// TwinCAT 3 PLC project PLC1
// ProgramVersion: 3.1.4024.12
// libraries:
//   Tc2_Standard, * (Beckhoff Automation GmbH)
//   Tc2_System, * (Beckhoff Automation GmbH)
//   Tc3_IPCDiag, * (Beckhoff Automation GmbH)
//   Tc3_JsonXml, * (Beckhoff Automation GmbH)
//   Tc3_Module, * (Beckhoff Automation GmbH)
// project tree:
//   / Class Diagram_Visitor.TcCD (not stored), PlcTask.TcTTO
//   FBs/Exporters/ FB_XmlExporter.TcPOU, FB_SysLogExporter.TcPOU
//   FBs/System Modules/ FB_Conveyor.TcPOU, FB_Heater.TcPOU, FB_IPCDiagnostics.TcPOU
//   ITFs/ I_SysModules.TcIO, I_Visitor.TcIO
//   POUs/ MAIN.TcPOU
// real-time tasks:
//   TASK PlcTask: cycle T#10ms, priority 20, ADS port 350

CONFIGURATION PLC1
    RESOURCE PLC ON TwinCAT3
        TASK PlcTask(INTERVAL := T#10ms, PRIORITY := 20);
        PROGRAM MAIN WITH PlcTask : MAIN;
    END_RESOURCE
END_CONFIGURATION

// ---- ITFs/I_SysModules.TcIO
INTERFACE I_SysModules

METHOD accept
VAR_INPUT
	iVisitor : I_Visitor;
END_VAR
END_METHOD

END_INTERFACE

// ---- ITFs/I_Visitor.TcIO
INTERFACE I_Visitor

METHOD visitConveyor
VAR_INPUT
	fbConveyor : FB_Conveyor;
END_VAR
END_METHOD

METHOD visitHeater
VAR_INPUT
	fbHeater : FB_Heater;
END_VAR
END_METHOD

METHOD visitIPC
VAR_INPUT
	fbIPC : FB_IPCDiagnostics;
END_VAR
END_METHOD

END_INTERFACE

// ---- POUs/MAIN.TcPOU
PROGRAM MAIN
VAR
	// Program Objects
	fbHeater			: ARRAY[0..2] OF FB_Heater;
	fbConveyor 			: ARRAY[0..1] OF FB_Conveyor;
	fbIPCDiagnostics 	: FB_IPCDiagnostics;
	iModules 			: ARRAY[0..5] OF I_SysModules := [fbHeater[0], fbHeater[1], fbHeater[2], fbConveyor[0],  fbConveyor[1], fbIPCDiagnostics];
	
	// Visitor Object Control
	exportVisitor 		: FB_SysLogExporter;
	exportXML			: FB_XmlExporter('C:\TwinCAT\Visitor.xml', 'CX-12345');
	
	// Demo Program Control
	bLogExport			: BOOL;
	bXmlExport			: BOOL;
	bExecSave			: BOOL;
	i					: INT;
END_VAR

// Export the Syslog
IF bLogExport THEN
	bLogExport := FALSE;
	FOR i := 0 TO 5 DO
		iModules[i].accept(exportVisitor);
	END_FOR
END_IF

// Export for XML
IF bXmlExport THEN
	bXmlExport := FALSE;
	FOR i := 0 TO 5 DO
		iModules[i].accept(exportXML);
	END_FOR
	bExecSave := TRUE;
END_IF

IF exportXML.saveDoc(bExec := bExecSave) THEN
	bExecSave := FALSE;
END_IF

END_PROGRAM

// ---- FBs/System Modules/FB_Heater.TcPOU
{attribute 'reflection'} 
FUNCTION_BLOCK FB_Heater IMPLEMENTS I_SysModules
VAR
	lrCurrentTemp : LREAL := 72.0;
	sStatus		  : STRING := 'Heating...';
	
	{attribute 'instance-path'} 
    {attribute 'noinit'} 
    sPath : STRING; 
END_VAR

METHOD accept
VAR_INPUT
	iVisitor : I_Visitor;
END_VAR
iVisitor.visitHeater(THIS^);
END_METHOD

PROPERTY pPath : STRING
GET
pPath := THIS^.sPath;
END_GET
END_PROPERTY

PROPERTY pStatus : STRING
GET
pStatus := THIS^.sStatus;
END_GET
END_PROPERTY

PROPERTY pTemp : LREAL
GET
pTemp := THIS^.lrCurrentTemp;
END_GET
END_PROPERTY

END_FUNCTION_BLOCK

// ---- FBs/System Modules/FB_Conveyor.TcPOU
{attribute 'reflection'} 
FUNCTION_BLOCK FB_Conveyor IMPLEMENTS I_SysModules
VAR
	lrVelocity 	: LREAL := 500.00;
	lrPosition 	: LREAL := 127.00;
	sStatus		: STRING := 'Running';
	
	{attribute 'instance-path'} 
    {attribute 'noinit'} 
    sPath : STRING; 
END_VAR

METHOD accept
VAR_INPUT
	iVisitor : I_Visitor;
END_VAR
iVisitor.visitConveyor(THIS^);
END_METHOD

PROPERTY pPath : STRING
GET
pPath := THIS^.sPath;
END_GET
END_PROPERTY

PROPERTY pPosition : LREAL
GET
pPosition := THIS^.lrPosition;
END_GET
END_PROPERTY

PROPERTY pStatus : STRING
GET
pStatus := THIS^.sStatus;
END_GET
END_PROPERTY

PROPERTY pVelocity : LREAL
GET
pVelocity := THIS^.lrPosition;
END_GET
END_PROPERTY

END_FUNCTION_BLOCK

// ---- FBs/System Modules/FB_IPCDiagnostics.TcPOU
{attribute 'reflection'} 
FUNCTION_BLOCK FB_IPCDiagnostics IMPLEMENTS I_SysModules
VAR
	nCpuTemperature	: INT := 75;	// CPU temperature [°F]
	nCpuUsage       : INT := 5;    // CPU usage [%]
	
	
	{attribute 'instance-path'} 
    {attribute 'noinit'} 
    sPath : STRING; 
END_VAR

METHOD accept
VAR_INPUT
	iVisitor : I_Visitor;
END_VAR
iVisitor.visitIPC(THIS^);
END_METHOD

PROPERTY pCPU_Temp : INT
GET
pCPU_Temp := THIS^.nCpuTemperature;
END_GET
END_PROPERTY

PROPERTY pCPU_Usage : INT
GET
pCPU_Usage := THIS^.nCpuUsage;
END_GET
END_PROPERTY

PROPERTY pPath : STRING
GET
pPath := THIS^.sPath;
END_GET
END_PROPERTY

END_FUNCTION_BLOCK

// ---- FBs/Exporters/FB_SysLogExporter.TcPOU
FUNCTION_BLOCK FB_SysLogExporter IMPLEMENTS I_Visitor
VAR_INPUT
END_VAR
VAR_OUTPUT
END_VAR
VAR
END_VAR

METHOD visitConveyor
VAR_INPUT
	fbConveyor : FB_Conveyor;
END_VAR
ADSLOGSTR( msgCtrlMask := ADSLOG_MSGTYPE_LOG, msgFmtStr := '', strArg := '');
ADSLOGSTR( msgCtrlMask := ADSLOG_MSGTYPE_LOG, msgFmtStr := 'PLC Msg. *** Printing Messages For: %s', strArg := fbConveyor.pPath);
ADSLOGSTR( msgCtrlMask := ADSLOG_MSGTYPE_LOG, msgFmtStr := CONCAT(fbConveyor.pPath,':: Status := %s'), strArg := TO_STRING(fbConveyor.pStatus));
ADSLOGSTR( msgCtrlMask := ADSLOG_MSGTYPE_LOG, msgFmtStr := CONCAT(fbConveyor.pPath,':: Velocity := %s'), strArg := TO_STRING(fbConveyor.pVelocity));
ADSLOGSTR( msgCtrlMask := ADSLOG_MSGTYPE_LOG, msgFmtStr := CONCAT(fbConveyor.pPath,':: Position := %s'), strArg := TO_STRING(fbConveyor.pPosition));
END_METHOD

METHOD visitHeater
VAR_INPUT
	fbHeater : FB_Heater;
END_VAR
ADSLOGSTR( msgCtrlMask := ADSLOG_MSGTYPE_LOG, msgFmtStr := '', strArg := '');
ADSLOGSTR( msgCtrlMask := ADSLOG_MSGTYPE_LOG, msgFmtStr := 'PLC Msg. *** Printing Messages For: %s', strArg := fbHeater.pPath);
ADSLOGSTR( msgCtrlMask := ADSLOG_MSGTYPE_LOG, msgFmtStr := CONCAT(fbHeater.pPath,':: Status := %s'), strArg := TO_STRING(fbHeater.pStatus));
ADSLOGSTR( msgCtrlMask := ADSLOG_MSGTYPE_LOG, msgFmtStr := CONCAT(fbHeater.pPath,':: Temperature := %s'), strArg := TO_STRING(fbHeater.pTemp));
END_METHOD

METHOD visitIPC
VAR_INPUT
	fbIPC : FB_IPCDiagnostics;
END_VAR
ADSLOGSTR( msgCtrlMask := ADSLOG_MSGTYPE_LOG, msgFmtStr := '', strArg := '');
ADSLOGSTR( msgCtrlMask := ADSLOG_MSGTYPE_LOG, msgFmtStr := 'PLC Msg. *** Printing Messages For: %s', strArg := fbIPC.pPath);
ADSLOGSTR( msgCtrlMask := ADSLOG_MSGTYPE_LOG, msgFmtStr := CONCAT(fbIPC.pPath,':: CPU Usage := %s'), strArg := TO_STRING(fbIPC.pCPU_Usage));
ADSLOGSTR( msgCtrlMask := ADSLOG_MSGTYPE_LOG, msgFmtStr := CONCAT(fbIPC.pPath,':: CPU Temperature (F) := %s'), strArg := TO_STRING(fbIPC.pCPU_Temp));
END_METHOD

END_FUNCTION_BLOCK

// ---- FBs/Exporters/FB_XmlExporter.TcPOU
FUNCTION_BLOCK FB_XmlExporter IMPLEMENTS I_Visitor
VAR
	sFilePath 		: STRING;
	sMachineName 	: STRING;	

	fbXml			: FB_XmlDomParser;
	objRoot 		: SXmlNode;
	objMachines 	: SXmlNode;
	objMachine		: SXmlNode;
	objModules		: SXmlNode;
	objModule		: SXmlNode;
	objAttribute 	: SXmlAttribute;
	sXmlString		: STRING(1000);
	nLength   		: UDINT;
END_VAR

METHOD FB_init : BOOL
VAR_INPUT
	bInitRetains 	: BOOL; // if TRUE, the retain variables are initialized (warm start / cold start)
	bInCopyCode 	: BOOL;  // if TRUE, the instance afterwards gets moved into the copy code (online change)
	sFilePath 		: STRING;
	sMachineName 	: STRING;
END_VAR
THIS^.sFilePath := sFilePath;
THIS^.sMachineName := sMachineName;

(* Create an empty XML document *)
objRoot := fbXml.GetDocumentNode();

(* Create a new XML node 'Machines' and add to the empty document *)
objMachines := fbXml.AppendNode(objRoot, 'Machines');

(* Create a new XML node 'Machine' and add an attribute to this node. Append node to 'Machines' *)
objMachine := fbXml.AppendNode(objMachines, 'Machine');
objAttribute := fbXml.AppendAttribute(objMachine, 'Name', sMachineName);

(* Create a new XML node 'Controllers' and add to the 'Machine' node *)
objModules := fbXml.AppendNode(objMachine, sMachineName);
END_METHOD

METHOD saveDoc : BOOL
VAR_INPUT
	bExec : BOOL;
END_VAR
(* Retrieve XML document and store in a variable of data type STRING(1000) *)
nLength := fbXml.CopyDocument(sXmlString, SIZEOF(sXmlString));

SaveDoc := fbXml.SaveDocumentToFile(sFile := THIS^.sFilePath, bExec := bExec);
END_METHOD

METHOD visitConveyor
VAR_INPUT
	fbConveyor : FB_Conveyor;
END_VAR
VAR
	Path : STRING;
	Position : STRING;
	Velocity : STRING;
	Status : STRING;
END_VAR
Path := fbConveyor.pPath;
Position := TO_STRING(fbConveyor.pPosition);
Velocity := TO_STRING(fbConveyor.pVelocity);
Status := fbConveyor.pStatus;

objModule := fbXml.AppendChild(objModules, 'Conveyor', Path, FALSE);
objAttribute := fbXml.AppendAttribute(objModule, 'Position', Position);
objAttribute := fbXml.AppendAttribute(objModule, 'Velocity', Velocity);
objAttribute := fbXml.AppendAttribute(objModule, 'Status', Status);
END_METHOD

METHOD visitHeater
VAR_INPUT
	fbHeater : FB_Heater;
END_VAR
VAR
	Path : STRING;
	Temp : STRING;
	Status : STRING;
END_VAR
Path := fbHeater.pPath;
Temp := TO_STRING(fbHeater.pTemp);
Status := fbHeater.pStatus;

objModule := fbXml.AppendChild(objModules, 'Heater', Path, FALSE);
objAttribute := fbXml.AppendAttribute(objModule, 'Temperature', Temp);
objAttribute := fbXml.AppendAttribute(objModule, 'Status', Status);
END_METHOD

METHOD visitIPC
VAR_INPUT
	fbIPC : FB_IPCDiagnostics;
END_VAR
VAR
	Path : STRING;
	CPU_Temp : STRING;
	CPU_Usage : STRING;
END_VAR
Path := fbIPC.pPath;
CPU_Temp := TO_STRING(fbIPC.pCPU_Temp);
CPU_Usage := TO_STRING(fbIPC.pCPU_Usage);

objModule := fbXml.AppendChild(objModules, 'IPC_Diagnostics', Path, FALSE);
objAttribute := fbXml.AppendAttribute(objModule, 'CPU_Temperature', CPU_Temp);
objAttribute := fbXml.AppendAttribute(objModule, 'CPU_Usage', CPU_Usage);
END_METHOD

END_FUNCTION_BLOCK
